ABB RobotStudio station: Proyecto_Prog_Robots_1.rsstnx

Station Proyecto_Prog_Robots (saved by RobotStudio 23.2.10395.0)
Controller thethirdone, task T_ROB1: task frame (RAPID world) sits at (1989.62, -993.99, 775) mm, rotated rx 0 ry 0 rz 90 deg in the station
Controller thesecondone, task T_ROB1: task frame (RAPID world) sits at (1997.05, 1000.95, 775) mm, rotated rx 0 ry 0 rz -90 deg in the station
Controller themainone, task T_ROB1: task frame (RAPID world) sits at (0, 0, 775) mm, rotated rx 0 ry 0 rz 180 deg in the station
Controller themainone
  mechanical unit ROB_1: themainone, 6 joints, base frame (0, 0, 0) mm
Controller thesecondone
  mechanical unit ROB_1: thesecondone, 6 joints, base frame (0, 0, 0) mm
Controller thethirdone
  mechanical unit ROB_1: thethirdone, 6 joints, base frame (0, 0, 0) mm
Layout (positions relative to the parent item):
  - themainone [mechanism, from %ABB.RobotStudio.Models.IRB120%\IRB120_3_58_G_01.rslib] at (0, 0, 775) mm, rotated rx 0 ry 0 rz 180 deg; joint values [0.243, 0.7605, -0.6077, 0, 0.5484, 0.243] (rad or m)
  - thesecondone [mechanism, from %ABB.RobotStudio.Models.IRB120%\IRB120_3_58_G_01.rslib] at (1997.05, 1000.95, 775) mm, rotated rx 0 ry 0 rz -90 deg; joint values [0, 0, 0, 0, 0.5236, 0] (rad or m)
  - thethirdone [mechanism, from %ABB.RobotStudio.Models.IRB120%\IRB120_3_58_G_01.rslib] at (1989.62, -993.99, 775) mm, rotated rx 0 ry 0 rz 90 deg; joint values [0, 0, 0, 0, 0.5236, 0] (rad or m)
  - conveyor_2 [part, from %ABB.RobotStudio.Models.Conveyors%\Conveyor Guide 400.rslib] at (-300, -660, 0) mm
  - conveyor_3 [part, from %ABB.RobotStudio.Models.Conveyors%\Conveyor Guide 400.rslib] at (-300, 250, 0) mm
  - soport_1 [part], size 300 x 299.2 x 725 mm
  - sop_1 [part] at (0, 0, 725) mm, size 360 x 358 x 50 mm
  - soport_2 [part] at (1997.05, 1000.95, 0) mm, size 350 x 349.2 x 725 mm
  - sop_2 [part] at (1997.05, 1000.95, 725) mm, size 380 x 377.9 x 50 mm
  - soport_3 [part] at (1989.62, -993.99, 0) mm, size 350 x 349.2 x 725 mm
  - sop_3 [part] at (1989.62, -993.99, 725) mm, size 380 x 377.9 x 50 mm
  - TOOL [smart component]
      signals: DI COGER8, DI SOLTAR
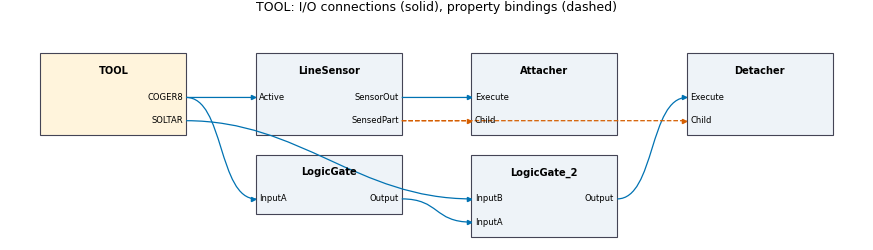
      connections:
        LineSensor.SensorOut -> Attacher.Execute
        TOOL.COGER8 -> LineSensor.Active
        TOOL.COGER8 -> LogicGate.InputA
        TOOL.SOLTAR -> LogicGate_2.InputB
        LogicGate.Output -> LogicGate_2.InputA
        LogicGate_2.Output -> Detacher.Execute
        LineSensor.SensedPart => Attacher.Child
        LineSensor.SensedPart => Detacher.Child
    - Gripper [mechanism] at (-534.1, -132.39, 1237.34) mm, rotated rx 164.1 ry 47.86 rz -7.09 deg
        TCP Gripper at (0, 0, 50) mm
        links: VacuumGripperDefinitivo_3
    - Attacher [smart component, from Components\Attacher.rslib]
        properties: Parent=Gripper; Flange=0; Child=(none); Mount=false; Offset=[0 0 0]; Orientation=[0 0 0]
    - Detacher [smart component, from Components\Detacher.rslib]
        properties: Child=(none); KeepPosition=true
    - LineSensor [smart component, from Components\LineSensor.rslib] at (-572.13, -141.88, 1203.96) mm, rotated rx -164.1 ry -47.86 rz 172.91 deg
        properties: Start=[0 0 0]; End=[0 0 0.015]; Length=0.015; Radius=0.00135135135135135; Tag=(none); SensedPart=(none); SensedPoint=[-0.06480419921875 -0.464987457275391 0.843276123046875]
      - _sensorPart_ [part], size 2.7 x 2.7 x 15 mm
    - LogicGate [smart component, from Components\LogicGate.rslib]
        properties: Operator=NOT; Delay=0
    - LogicGate_2 [smart component, from Components\LogicGate.rslib]
        properties: Operator=AND; Delay=0
  - Cinta transportadora_2 [smart component]
      signals: DI EncenderMotor, DO Headphones_Sensor, DO Mouse_Sensor, DI Reset_Mouse
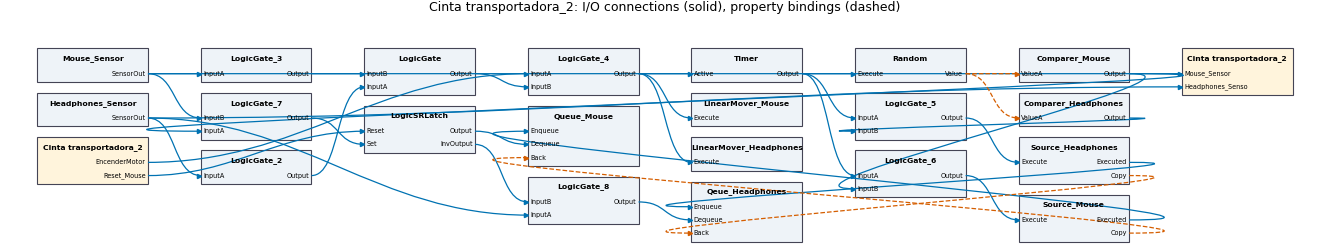
      connections:
        Mouse_Sensor.SensorOut -> Cinta transportadora_2.Mouse_Sensor
        Headphones_Sensor.SensorOut -> Cinta transportadora_2.Headphones_Sensor
        Source_Headphones.Executed -> Qeue_Headphones.Enqueue
        Source_Mouse.Executed -> Queue_Mouse.Enqueue
        Mouse_Sensor.SensorOut -> LogicGate_3.InputA
        LogicGate_3.Output -> LogicGate.InputB
        Headphones_Sensor.SensorOut -> LogicGate_2.InputA
        LogicGate_2.Output -> LogicGate.InputA
        Cinta transportadora_2.EncenderMotor -> LogicGate_4.InputA
        LogicGate.Output -> LogicGate_4.InputB
        LogicGate_4.Output -> Timer.Active
        Timer.Output -> Random.Execute
        Timer.Output -> LogicGate_5.InputA
        Timer.Output -> LogicGate_6.InputA
        Comparer_Mouse.Output -> LogicGate_6.InputB
        Comparer_Headphones.Output -> LogicGate_5.InputB
        LogicGate_4.Output -> LinearMover_Mouse.Execute
        LogicGate_4.Output -> LinearMover_Headphones.Execute
        LogicGate_5.Output -> Source_Headphones.Execute
        LogicGate_6.Output -> Source_Mouse.Execute
        Cinta transportadora_2.Reset_Mouse -> LogicSRLatch.Reset
        LogicGate_7.Output -> LogicSRLatch.Set
        LogicGate_8.Output -> Qeue_Headphones.Dequeue
        Mouse_Sensor.SensorOut -> LogicGate_7.InputB
        LogicSRLatch.Output -> Queue_Mouse.Dequeue
        LogicSRLatch.InvOutput -> LogicGate_8.InputB
        Headphones_Sensor.SensorOut -> LogicGate_8.InputA
        Comparer_Mouse.Output -> LogicGate_7.InputA
        Source_Headphones.Copy => Qeue_Headphones.Back
        Source_Mouse.Copy => Queue_Mouse.Back
        Random.Value => Comparer_Mouse.ValueA
        Random.Value => Comparer_Headphones.ValueA
    - conveyor_1 [part, from %ABB.RobotStudio.Models.Conveyors%\Conveyor Guide 400.rslib] at (-3350, -210, 0) mm
    - Headphones_Box [part], size 250 x 250 x 125 mm
    - Mouse_Box [part], size 170 x 120 x 75 mm
    - Headphones_Sensor [smart component, from Components\LineSensor.rslib] at (-482.73, 129.96, 892.43) mm, rotated rx 90 ry 0 rz 0 deg
        properties: Start=[0 0 0]; End=[0 0 0.3]; Length=0.3; Radius=0; Tag=(none); SensedPart=(none); SensedPoint=[-0.482727294921875 0.0999999923706055 0.892429992675781]
      - _sensorPart_ [part], size 0 x 0 x 300 mm
    - Mouse_Sensor [smart component, from Components\LineSensor.rslib] at (-482.73, 129.96, 820.43) mm, rotated rx 90 ry 0 rz 0 deg
        properties: Start=[0 0 0]; End=[0 0 0.3]; Length=0.3; Radius=0; Tag=(none); SensedPart=(none); SensedPoint=[-0.48272705078125 0.0999999923706055 0.820429992675781]
      - _sensorPart_ [part], size 0 x 0 x 300 mm
    - Source_Mouse [smart component, from Components\Source.rslib]
        properties: Source=Mouse_Box; Copy=(none); Parent=(none); Position=[0 0 0]; Orientation=[0 0 0]; Transient=true; PhysicsBehavior=-1
    - Source_Headphones [smart component, from Components\Source.rslib]
        properties: Source=Headphones_Box; Copy=(none); Parent=(none); Position=[0 0 0]; Orientation=[0 0 0]; Transient=true; PhysicsBehavior=-1
    - Qeue_Headphones [smart component, from Components\Queue.rslib]
        properties: Back=(none); Front=(none); Queue={7c6882b9-f051-4767-a359-e968a9221f25};{30578bb3-0eb2-425d-acb6-8b23693ebdb2};{d97f1cd3-a2f7-4bd6-92b9-76b3eb2b6e34};{c300db59-31d5-4efb-b1e8-bc170c6ecb60};{2232bca8-2d3f-4403-8a8e-013e99c0ff53};{23439bc7-5991-49e0-b46d-990f1ae2c20c};{cc20a378-5d0a-4886-9283-99e369d1a319};{0abf2617-e11c-4108-92e6-09a6a8a73df5};{eb6215ba-01f3-4f6a-af7b-b096765bc1a0};{f8c40b83-5b43-4230-a074-1abcf6cb5528};{ac9cfbe9-b626-40c0-a955-5efb1156dd65};{c17f1e12-160d-4a9a-bfbd-9d127e26952b};{87c1d730-25e3-4d95-bf46-2ce6953c0a7a};{471a3580-2351-4f02-b6d5-f27bd4d19176};{7185d0c9-903b-4160-b2c7-79e85702f161};{51bb0b32-e131-4b79-be13-244167ea6728};{fb374b99-278f-4042-80c8-4ff4606e81e9};{df820581-4cbe-4353-9d5d-33283584515e};{e00e34a4-f45f-47e8-8181-a3d50d1ac628};{78632a17-2a19-4edd-8847-f6b4c8d83460};{84a30c24-7c0b-4b65-ac37-99b44562191a};{8027a2b4-e236-4952-84fe-1eb643f80800};{5805a7cd-0d46-4e7d-bdc9-88d240ed65b7};{1f151e77-ded0-4d51-8fd4-a2fa48a39306};{03953787-ae18-43b5-a33f-45b4e9c5ab71};{21698db0-4a52-4c80-9362-9db08066e000};{5ade8c01-4537-4928-8a26-9fb68819b8f8};{99af3ad3-4df6-4c0d-a1be-ab3bdc90e27b};{f730e1e6-1a94-4632-ad1d-0bbe29b6e37b};{6e637696-44d8-4e58-afc3-34cedaf88940};{029cdd1a-de1e-43a0-bd3e-6ff29247f429};{aab67a26-d2d3-450b-9cb3-37c84193c221};{f524097d-fd21-48cc-9eff-77c752a61cb9};{5be0302b-507e-49a1-853d-f488945db40d};{1e3a02bb-5e1e-4921-bffa-0abd8b2c81ce};{a0d16ae2-cec9-41e8-b227-04480e8508a6};{68126d46-cd9b-42bf-b6ca-0aad88b64699};{1ac53a62-2a29-4de9-91d4-edc6cbf9c9c9};{f57d71e0-093b-4d0d-b58b-55300de68e89};{e2bf03ca-ad4b-430f-824c-3fabefef1919};{92e476e6-88cd-4c01-8f89-da562d56f7e3};{2020d39d-c095-40c3-985b-1caca22e82d6};{d2ff7958-ba34-48b1-97b1-8bbeed3537f0};{526cc441-d97d-45c6-a8a6-ed8d0b60faf0};{9f5c79b0-7fbf-4379-ae8b-db2109dd0a88};{2cfa8728-08ed-49df-953e-644a74c5caf9};{fa55c1d9-fdb1-4fa1-a871-51ea5d9d0754};{a5fc95cb-68cb-456f-bc34-e5fa3b32cb98};{445a4aa4-fb09-4e45-bd6d-b9843f0c0f0a};{e62f2b0a-a484-497f-9b8c-8b889aca3682};{f49e6408-8b8d-4c59-8dda-bfebc9abd4e3};{5843614a-b41b-4084-a8aa-bbce56332b81};{c42f6e2c-8893-492f-adf7-7b8af2094e98};{4fb29d44-7d0b-4ed9-abea-593dc17932aa};{6ad027f1-2981-4a39-bd87-b8952a8667a2};{22f3cb03-bd8d-4bb3-97f0-573ee4a36f66};{b4e6f9d8-6a68-4200-9123-f649efdf29dc};{572a55f8-d922-4e25-9d42-c07cdd7eee04};{e6ddb73f-d1cf-4517-b020-a5fdef8584c0};{8a498a62-a7d3-4135-bb11-171ca7415efe};{190a5703-773a-406c-b9f7-5daeb07cf16c};{05c61745-b603-454a-9bdf-7efcff5d11ab}; NumberOfObjects=2
    - Queue_Mouse [smart component, from Components\Queue.rslib]
        properties: Back=(none); Front=(none); Queue={77e8c259-785c-4da3-81f7-99f189588a4e};{88174d8b-5cbc-4e98-a8c8-33c04d38a2ca};{8fc0be2f-e7d4-4778-88a7-7b118e6c2de8};{063506f1-bc05-49a7-9625-d5d7a89d171e};{869f6169-061b-4734-9e82-ad43ebfc7cbb};{ab2e570f-081e-414b-94ac-799cb4d5ae27};{c8719fd6-a68d-4bef-9b8f-32e14a0136bd};{9576c5fc-04e1-4edb-bc16-ea3777c66d84};{45c6b65e-216b-46af-ab0d-a6dfd0885c98};{e4294346-dce0-461f-bcca-a4ba9626d776};{c14c9ae6-2907-44f7-951c-852e0194cc7b};{2cb446c1-1b7b-4658-a6bd-c61ebc6e28cd};{a1c44c06-ea4d-4e31-9fce-db6260c64e39};{a0218873-9d05-425c-98a9-0bd4798d8de8};{771bfe29-d0b6-4166-8e45-5891340f6edd};{0dcca1ab-4586-4d6f-af1c-3ef883d51e9e};{c3df0daa-855e-4adc-8387-4830794cc92a};{e85743aa-88b6-419e-bc03-2e3516ef18de};{dde63b02-08b9-43a7-a746-f0d7627fd38e};{6e1e839f-b034-45a6-872e-758ddc7a3981};{7f1e5f8f-8331-4028-8c35-48d7db5d6f8c};{5efc2b13-ba29-4d03-a1cf-3708d0161bb1};{5d2b6413-8401-4dbb-93ce-fef1feb2883d};{5ecab99c-dc82-41e7-bde0-2ab61f5f0575};{9d444e73-c89d-4ecc-b44e-b34319035bc8};{00e78e6c-90d4-40d9-ab66-1d7a5fbb2c63};{72e9bb6b-3ad6-4e05-ac7d-78868f8e513f};{b45e3568-6646-4085-ad8f-a4b00a01c1f2};{d6284561-d7c3-426c-951e-47535ae9dffe};{1dfefc07-4a8b-4072-86eb-a7ae7fe97c84};{92d281df-96f6-4ff8-8ffe-406ce6f97e97};{b1965837-ef22-4bb6-8977-6479c5579d3e};{14870676-b05a-441b-b328-181318419b4d};{94dc42f2-2033-4f79-bc97-a94fe28f62ea};{fa51c0f7-7c91-4821-ae87-8b5c4a0f9bf4};{b5f5b61b-4f80-4808-b3c2-5e2393c2223f};{6e129c37-7602-44f3-b0b2-c66eac675676};{d3981c8c-bf4a-4fda-b72d-2f784a2f3dd3};{f755878a-11a2-48a9-b01d-4c58af847ba2}; NumberOfObjects=1
    - Timer [smart component, from Components\Timer.rslib]
        properties: StartTime=0; Interval=3; Repeat=true; CurrentTime=32.352
    - LogicGate [smart component, from Components\LogicGate.rslib]
        properties: Operator=AND; Delay=0
    - LogicGate_2 [smart component, from Components\LogicGate.rslib]
        properties: Operator=NOT; Delay=0
    - LogicGate_3 [smart component, from Components\LogicGate.rslib]
        properties: Operator=NOT; Delay=0
    - LogicGate_4 [smart component, from Components\LogicGate.rslib]
        properties: Operator=AND; Delay=0
    - Random [smart component, from Components\Random.rslib]
        properties: Value=0.176275516942272; Min=0; Max=1
    - Comparer_Headphones [smart component, from Components\Comparer.rslib]
        properties: ValueA=0.176275516942272; Operator=<=; ValueB=0.5
    - Comparer_Mouse [smart component, from Components\Comparer.rslib]
        properties: ValueA=0.176275516942272; Operator=>; ValueB=0.5
    - LogicGate_5 [smart component, from Components\LogicGate.rslib]
        properties: Operator=AND; Delay=0
    - LogicGate_6 [smart component, from Components\LogicGate.rslib]
        properties: Operator=AND; Delay=0
    - LinearMover_Mouse [smart component, from Components\LinearMover.rslib]
        properties: Object=Queue_Mouse; Direction=[3 0 0]; Speed=0.2; Reference=Global; ReferenceObject=(none)
    - LinearMover_Headphones [smart component, from Components\LinearMover.rslib]
        properties: Object=Qeue_Headphones; Direction=[3 0 0]; Speed=0.2; Reference=Global; ReferenceObject=(none)
    - LogicGate_7 [smart component, from Components\LogicGate.rslib]
        properties: Operator=AND; Delay=0
    - LogicGate_8 [smart component, from Components\LogicGate.rslib]
        properties: Operator=AND; Delay=0
    - LogicSRLatch [smart component, from Components\LogicSRLatch.rslib]
Attachment: Gripper is attached to themainone / Link6
Attachment: LineSensor is attached to Gripper / VacuumGripperDefinitivo_3
Station signals: DI empezar
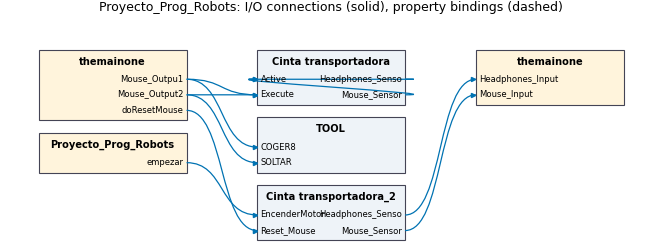
Station logic (signal -> signal, property => property):
  Cinta transportadora.Headphones_Sensor -> LineSensor.Active
  Cinta transportadora.Mouse_Sensor -> LineSensor_2.Active
  themainone.Mouse_Outpu1 -> Attacher_2.Execute
  themainone.Mouse_Output2 -> Detacher.Execute
  themainone.Mouse_Outpu1 -> TOOL.COGER8
  themainone.Mouse_Output2 -> TOOL.SOLTAR
  Proyecto_Prog_Robots.empezar -> Cinta transportadora_2.EncenderMotor
  Cinta transportadora_2.Headphones_Sensor -> themainone.Headphones_Input
  Cinta transportadora_2.Mouse_Sensor -> themainone.Mouse_Input
  themainone.doResetMouse -> Cinta transportadora_2.Reset_Mouse
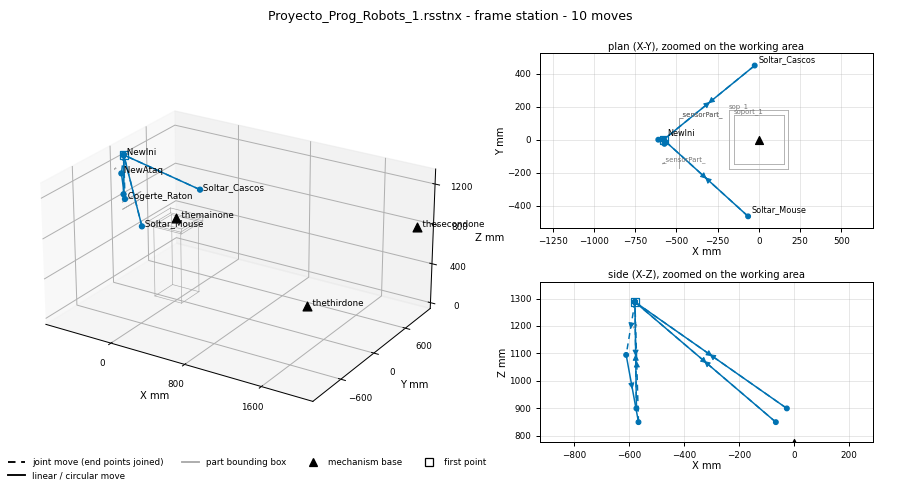
[picture p0: tool path of Proyecto_Prog_Robots_1.rsstnx in frame station, 10 of 10 moves have a stored position in this frame; points joined in program order, loops and branches not executed]
Targets, tools, work objects and paths stored in the station, written as RAPID:
! task T_ROB1
MODULE CalibData
  PERS tooldata MyTool:=[TRUE,[[31.792631019,0,229.638935148],[0.945518576,0,0.325568154,0]],[1,[0,0,1],[1,0,0,0],0,0,0]];
  TASK PERS wobjdata WO_themainone:=[FALSE,TRUE,"",[[0,0,0],[1,0,0,0]],[[0,0,0],[1,0,0,0]]];
  PERS tooldata VacuumGripper:=[TRUE,[[0,0,110],[1,0,0,0]],[1,[0,0,1],[1,0,0,0],0,0,0]];
  PERS tooldata Gripper:=[TRUE,[[0,0,50],[1,0,0,0]],[1,[0,0,1],[1,0,0,0],0,0,0]];
ENDMODULE

! task T_ROB1
MODULE Module1
  CONST robtarget NewIni:=[[577.89485234,0,512.371659812],[0.499999865,0,0.866025482,0],[0,0,0,0],[9E+09,9E+09,9E+09,9E+09,9E+09,9E+09]];
  CONST robtarget NewAtaq:=[[609.844394291,0,319.671174559],[0.430026102,0,0.902816455,0],[0,0,0,0],[9E+09,9E+09,9E+09,9E+09,9E+09,9E+09]];
  CONST robtarget Cogerte_Raton:=[[565,15,75],[0,0,1,0],[0,0,0,0],[9E+09,9E+09,9E+09,9E+09,9E+09,9E+09]];
  CONST robtarget Cogerte_Cascos:=[[572.555351259,25,125],[0,1,0,0],[0,0,-2,0],[9E+09,9E+09,9E+09,9E+09,9E+09,9E+09]];
  CONST robtarget Soltar_Cascos:=[[25,-450,125],[0,0,1,0],[-1,0,-1,0],[9E+09,9E+09,9E+09,9E+09,9E+09,9E+09]];
  CONST robtarget Soltar_Mouse:=[[65,465,75],[0,0,1,0],[0,0,0,0],[9E+09,9E+09,9E+09,9E+09,9E+09,9E+09]];
  PROC main()
    SetDO Mouse_Outpu1,0;
    SetDO Mouse_Output2,1;
    SetDO doResetMouse,1;
    SetDO doResetMouse,0;
    SetDO doResetMouse,0;
    MoveL NewIni,v1000,fine,Gripper\WObj:=WO_themainone;
    MoveJ NewAtaq,v1000,fine,Gripper\WObj:=WO_themainone;
    WaitDI Mouse_Input,1;
    MoveL Cogerte_Raton,v1000,fine,Gripper\WObj:=WO_themainone;
    SetDO Mouse_Output2,0;
    SetDO Mouse_Outpu1,1;
    SetDO doResetMouse,1;
    MoveJ NewIni,v1000,fine,Gripper\WObj:=WO_themainone;
    MoveL Soltar_Mouse,v1000,fine,Gripper\WObj:=WO_themainone;
    SetDO Mouse_Outpu1,0;
    SetDO Mouse_Output2,1;
    MoveJ NewIni,v1000,fine,Gripper\WObj:=WO_themainone;
    MoveL Cogerte_Cascos,v1000,fine,Gripper\WObj:=WO_themainone;
    SetDO Mouse_Output2,0;
    SetDO Mouse_Outpu1,1;
    MoveJ NewIni,v1000,fine,Gripper\WObj:=WO_themainone;
    MoveL Soltar_Cascos,v1000,fine,Gripper\WObj:=WO_themainone;
    SetDO Mouse_Outpu1,0;
    SetDO Mouse_Output2,1;
    MoveJ NewIni,v1000,fine,Gripper\WObj:=WO_themainone;
  ENDPROC
ENDMODULE

! task T_ROB1
MODULE CalibData
  PERS tooldata MyTool:=[TRUE,[[31.792631019,0,229.638935148],[0.945518576,0,0.325568154,0]],[1,[0,0,1],[1,0,0,0],0,0,0]];
ENDMODULE

! task T_ROB1
MODULE CalibData
  PERS tooldata MyTool:=[TRUE,[[31.792631019,0,229.638935148],[0.945518576,0,0.325568154,0]],[1,[0,0,1],[1,0,0,0],0,0,0]];
ENDMODULE

